INTERFACE I_XTS

METHOD AreAllMoversStationary : BOOL
END_METHOD

METHOD DisableXTS : BOOL
VAR_INPUT
END_VAR
END_METHOD

METHOD EnableXTS : BOOL
VAR_INPUT
END_VAR
END_METHOD

METHOD GetErrorCode : UDINT
VAR_INPUT
END_VAR
END_METHOD

METHOD HasError : BOOL
VAR_INPUT
END_VAR
END_METHOD

PROPERTY Initialised : BOOL
GET
END_GET
END_PROPERTY

METHOD IsXtsIdle : BOOL
VAR_INPUT
END_VAR
END_METHOD

METHOD IsXtsReady : BOOL
VAR_INPUT
END_VAR
END_METHOD

METHOD PUBLIC Abstract MoverHomeSequence : BOOL
VAR_INPUT
END_VAR
END_METHOD

METHOD RegisterMovers : HRESULT
VAR_INPUT
	MyMover : I_XtsMover;
END_VAR
END_METHOD

METHOD Reset : BOOL
VAR_INPUT
END_VAR
END_METHOD

METHOD StopXts : BOOL
VAR_INPUT
END_VAR
END_METHOD

END_INTERFACE

(* stored: Version 1.1.0.1
   Itf I_XTS: Id {eb22a7d8-6cc9-41fe-bacb-ecb9c288212d}
   Folder Operations: Id {fcac5daf-610f-4795-a9df-a1a0b59d368f}
   Folder Status: Id {e945740f-30ab-470b-b703-ee9e691fdeff}
   Method AreAllMoversStationary: Id {b214b570-8dd1-4577-80c2-923199586750}
   Method DisableXTS: Id {d730e6bc-30f4-400f-83c5-0a8ef7530dc6}
   Method EnableXTS: Id {a90bf243-5fbb-42eb-a2e5-eb1ea9f490a9}
   Method GetErrorCode: Id {8d18bfb1-883b-4192-b6c9-acf73a59bec9}
   Method HasError: Id {af275816-6e74-427c-9fdf-440990004afa}
   Property Initialised: Id {29344615-27fb-4ea5-ad7a-fc8898059767}
   Get Get: Id {57975104-c7c3-4f8a-9853-70129e27cdaf}
   Method IsXtsIdle: Id {a58467b2-fd55-49b7-9538-35b2ad34103b}
   Method IsXtsReady: Id {88e988d8-b3fd-4023-a27f-e2263614dcbf}
   Method MoverHomeSequence: Id {80de9bd3-37be-4579-86bc-1293deec4463}
   Method RegisterMovers: Id {e65bc655-b1b5-4ed3-91eb-2d51871a4d75}
   Method Reset: Id {1314f0dc-0a66-4dbc-aa58-dd78d21ed251}
   Method StopXts: Id {d7591d56-8a8c-46a1-bfd3-85f1f168760d} *)
